(* PLC project mtcs_m2, Institute of Astronomy OntoManager 0.0.1 *)
(* stored: creationDateTime 2017-02-03T09:55:41.735679, modificationDateTime 2017-02-03T09:55:41.735679 *)

TYPE M2Axes : (X := 0, Y := 1, Z := 2, TILTX := 3, TILTY := 4);
END_TYPE

TYPE M2MoveProcedureStates : (IDLE := 0, ABORTED := 1, PREPARE_PROCESS := 2, MOVING := 3, MOVING_TO_ANTI_BACKLASH_POSITION := 4, MOVING_CLOSE_TO_FINAL_POSITION := 5, MOVING_TO_FINAL_POSITION := 6, ERROR := 7, ABORTING := 8);
END_TYPE

TYPE M2Parts : STRUCT
  powerRelay : SimpleRelay;  (* Relay to power on/off the power of the M2 field electricity *)
  heater : SimpleRelay;  (* Digital output to power on/off the heater of M2 *)
  x : M2XAxis;  (* The X axis *)
  y : M2YAxis;  (* The Y axis *)
  z : M2ZAxis;  (* The Z axis *)
  tiltX : M2TiltXAxis;  (* The TiltX axis *)
  tiltY : M2TiltYAxis;  (* The TiltY axis *)
  multiplexer : M2Multiplexer;  (* The multiplexer inputs and outputs *)
  configManager : ConfigManager;  (* The config manager (to load/save/activate configuration data) *)
  moveStepsProcedure : M2MoveStepsProcedure;  (* The move steps procedure *)
  movePositionProcedure : M2MovePositionProcedure;  (* The move to a certain position procedure *)
END_STRUCT;
END_TYPE

TYPE M2MultiplexerParts : STRUCT
  A : SimpleRelay;  (* Output A of the multiplexer corresponding with the selected axis *)
  B : SimpleRelay;  (* Output B of the multiplexer corresponding with the selected axis *)
  C : SimpleRelay;  (* Output C of the multiplexer corresponding with the selected axis *)
  driveEnable : SimpleRelay;  (* Enabled (TRUE) if the drive selected by the multiplexer must be enabled, Disabled (FALSE) if it must be disabled *)
  CW : SimpleRelay;  (* Enabled (TRUE) if the motor selected by the multiplexer will run in CW direction (- motion on the screw), Disabled (FALSE) if it will run in CCW direction (+ motion on the screw) *)
  release : SimpleRelay;  (* Disabled (FALSE) if the motor selected by the multiplexer must be braking, Enabled (TRUE) if it must be released *)
END_STRUCT;
END_TYPE

TYPE M2ZAxisParts : STRUCT
  highSpeed : SimpleRelay;  (* Enabled (TRUE) to enable the high-speed motion of the Z axis, Disabled (FALSE) to leave it low-speed *)
  encoder : SSIEncoder;  (* The SSI encoder of the Z axis *)
END_STRUCT;
END_TYPE

TYPE M2Processes : STRUCT
  initialize : Process;  (* Start initializing *)
  lock : Process;  (* Lock the system *)
  unlock : Process;  (* Unlock the system *)
  changeOperatingState : ChangeOperatingStateProcess;  (* Change the operating state (e.g. AUTO, MANUAL, ...) *)
  moveAbsolute : M2MoveProcess;  (* Move the position of one axis in an absolute way *)
  moveRelative : M2MoveProcess;  (* Move the position of one axis relative to the current position *)
  moveSteps : M2MoveStepsProcess;  (* Move the position of one axis by providing a number of steps (i.e. motor pulses) *)
  doThermalFocus : Process;  (* Do a thermal focus for the currently active focus *)
  doThermalFocusForStationName : M2DoThermalFocusForStationName;  (* Do a thermal focus for a specified focal station (based on the configured name of the station) *)
  doThermalFocusForStationPosition : M2DoThermalFocusForStationPosition;  (* Do a thermal focus for a specified focal station (based on the station numerical ID) *)
  verifyFixedPositions : Process;  (* Verify (and adjust if necessary) the fixed positions of X, Y, TiltX, and TiltY *)
  powerOn : Process;  (* Power on the M2 electricity *)
  powerOff : Process;  (* Power off the M2 electricity *)
  abort : Process;  (* Abort the move procedure *)
END_STRUCT;
END_TYPE

TYPE M2MultiplexerProcesses : STRUCT
  selectAxis : M2SelectAxisProcess;  (* Select an axis *)
END_STRUCT;
END_TYPE

TYPE M2Statuses : STRUCT
  initializationStatus : InitializationStatus;
  poweredStatus : PoweredStatus;
  healthStatus : HealthStatus;
  busyStatus : BusyStatus;
  operatingStatus : OperatingStatus;
END_STRUCT;
END_TYPE

TYPE M2MultiplexerStatuses : STRUCT
  healthStatus : HealthStatus;  (* Is the selected drive healthy? *)
  busyStatus : BusyStatus;  (* Is the selected drive busy? *)
END_STRUCT;
END_TYPE

TYPE M2XAxisStatuses : STRUCT
  healthStatus : HealthStatus;  (* Is the axis healthy? *)
END_STRUCT;
END_TYPE

TYPE M2YAxisStatuses : STRUCT
  healthStatus : HealthStatus;  (* Is the axis healthy? *)
END_STRUCT;
END_TYPE

TYPE M2TiltXAxisStatuses : STRUCT
  healthStatus : HealthStatus;  (* Is the axis healthy? *)
END_STRUCT;
END_TYPE

TYPE M2TiltYAxisStatuses : STRUCT
  healthStatus : HealthStatus;  (* Is the axis healthy? *)
END_STRUCT;
END_TYPE

TYPE M2ZAxisStatuses : STRUCT
  healthStatus : HealthStatus;  (* Is the axis healthy? *)
END_STRUCT;
END_TYPE

TYPE M2MoveStepsProcedureStatuses : STRUCT
  busyStatus : BusyStatus;  (* Is the M2MoveStepsProcedure in a busy state? *)
  healthStatus : HealthStatus;  (* Is the M2MoveStepsProcedure in a healthy state? *)
END_STRUCT;
END_TYPE

TYPE M2MovePositionProcedureStatuses : STRUCT
  busyStatus : BusyStatus;  (* Is the M2MoveAbsoluteProcedure in a busy state? *)
  healthStatus : HealthStatus;  (* Is the M2MoveAbsoluteProcedure in a healthy state? *)
END_STRUCT;
END_TYPE

TYPE M2Config : STRUCT
  x : M2PotentiometerAxisConfig;  (* The config of the X axis *)
  y : M2PotentiometerAxisConfig;  (* The config of the Y axis *)
  z : M2ZAxisConfig;  (* The config of the Z axis *)
  tiltX : M2PotentiometerAxisConfig;  (* The config of the tiltX axis *)
  tiltY : M2PotentiometerAxisConfig;  (* The config of the tiltY axis *)
  thermalFocus : M2ThermalFocusConfig;  (* The thermal focus coefficients for all focal stations *)
  waitAfterPowerOn : LREAL;  (* Time (in seconds) to wait after the field electricity of M2 have been powered on *)
  waitAfterPowerOff : LREAL;  (* Time (in seconds) to wait after the field electricity of M2 have been powered off *)
  powerOffTimeout : LREAL;  (* If no new command is sent to M2 within this time (in seconds) after completion of the last command, M2 will be powered off automatically *)
  fixedXPosition : LREAL;  (* The fixed X position in mm *)
  fixedXPositionTolerance : LREAL;  (* If the X position is within fixedXPosition +/- this tolerance, there's no need to adjust it *)
  fixedYPosition : LREAL;  (* The fixed Y position in mm *)
  fixedYPositionTolerance : LREAL;  (* If the Y position is within fixedYPosition +/- this tolerance, there's no need to adjust it *)
  fixedTiltXPosition : LREAL;  (* The fixed TiltX position in mm *)
  fixedTiltXPositionTolerance : LREAL;  (* If the TiltX position is within fixedTiltXPosition +/- this tolerance, there's no need to adjust it *)
  fixedTiltYPosition : LREAL;  (* The fixed TiltY position in mm *)
  fixedTiltYPositionTolerance : LREAL;  (* If the TiltY position is within fixedTiltYPosition +/- this tolerance, there's no need to adjust it *)
  verifyFixedPositinsOnThermalFocus : BOOL;  (* Each time a theremal focus is done, verify the fixed positions (and adjust them if they fall out of the tolerance) *)
END_STRUCT;
END_TYPE

TYPE M2ThermalFocusStationConfig : STRUCT
  offset : LREAL;  (* focus = offset + topCoefficient*topTemperature + centreCoefficient*centreTemperature + mirrorCellCoefficient*mirrorCellTemperature *)
  topCoefficient : LREAL;  (* focus = offset + topCoefficient*topTemperature + centreCoefficient*centreTemperature + mirrorCellCoefficient*mirrorCellTemperature *)
  centreCoefficient : LREAL;  (* focus = offset + topCoefficient*topTemperature + centreCoefficient*centreTemperature + mirrorCellCoefficient*mirrorCellTemperature *)
  mirrorCellCoefficient : LREAL;  (* focus = offset + topCoefficient*topTemperature + centreCoefficient*centreTemperature + mirrorCellCoefficient*mirrorCellTemperature *)
END_STRUCT;
END_TYPE

TYPE M2ThermalFocusConfig : STRUCT
  cassegrain : M2ThermalFocusStationConfig;  (* Cassegrain thermal focus config *)
  nasmythA : M2ThermalFocusStationConfig;  (* Nasmyth A thermal focus config *)
  nasmythB : M2ThermalFocusStationConfig;  (* Nasmyth B thermal focus config *)
  nasmythC : M2ThermalFocusStationConfig;  (* Nasmyth C thermal focus config *)
  nasmythD : M2ThermalFocusStationConfig;  (* Nasmyth D thermal focus config *)
  other0 : M2ThermalFocusStationConfig;  (* Other 0 thermal focus config *)
  other1 : M2ThermalFocusStationConfig;  (* Other 1 thermal focus config *)
  other2 : M2ThermalFocusStationConfig;  (* Other 2 thermal focus config *)
  other3 : M2ThermalFocusStationConfig;  (* Other 3 thermal focus config *)
  other4 : M2ThermalFocusStationConfig;  (* Other 4 thermal focus config *)
END_STRUCT;
END_TYPE

TYPE M2AxisGeneralConfig : STRUCT
  measurement : MeasurementConfig;  (* Configure the position measurement *)
  stoppingSteps : UDINT;  (* The number of steps to be expected between the time at which the PLC realizes that the brake release signal must be set, and the time that the axis is fully stopped (for Z axis: at low speed) *)
  finalSenseCW : BOOL;  (* TRUE if the motor final sense must be ClockWise (- motion on the screw), FALSE if the motor final sense must be CounterClockWise (+ motion on the screw) (for Z axis: at low speed) *)
  closePosition : UDINT;  (* The number of steps between the Close position (C) and final position (F) *)
  antiBacklashPosition : UDINT;  (* The number of steps between the Anti-backlash position (A) and final position (F) *)
  waitAfterMove : LREAL;  (* Time (in seconds) to wait after the axis has been moved *)
  timeout : LREAL;  (* Timeout for a movement, in seconds (for Z-axis: at low speed) *)
END_STRUCT;
END_TYPE

TYPE M2ZAxisConfig : STRUCT
  general : M2AxisGeneralConfig;  (* Settings which are general for all axes *)
  highSpeedStoppingSteps : UDINT;  (* The number of steps to be expected between the time at which the PLC realizes that the brake release signal must be set, and the time that the axis is fully stopped at high speed *)
  highSpeedTimeout : LREAL;  (* Timeout for a fast movement of the Z axis (in seconds) *)
END_STRUCT;
END_TYPE

TYPE M2PotentiometerAxisConfig : STRUCT
  general : M2AxisGeneralConfig;  (* Settings which are general for all axes *)
  voltageCorrectionFactor : LREAL;  (* Position = voltage * correctionFactor * voltageToPosition *)
END_STRUCT;
END_TYPE

TYPE M2ConstantsZ : STRUCT
  MOT_TO_RED_RATIO : LREAL := 134.0;  (* Motor reduction ratio *)
  RED_TO_SCREW_RATIO : LREAL := 2.0;  (* Transmission ratio between the motor reduction and the screw *)
  SCREW_TO_ENC_RATIO : LREAL := 1.0;  (* Transmission ratio between the encoder and the screw *)
  MIN_POSITION : LREAL := 0.0;  (* Minimum position of the axis, in micrometer *)
  MAX_POSITION : LREAL := 50000.0;  (* Maximum position of the axis, in micrometer *)
  SCREW_PITCH : LREAL := 2000.0;  (* Screw pitch, in micrometer *)
  FEEDBACK_RESOLUTION : LREAL := 32;  (* Motor feedback resolution (pulses per revolution of the motor rotor) *)
END_STRUCT;
END_TYPE

TYPE M2ConstantsX : STRUCT
  MOT_TO_RED_RATIO : LREAL := 415.0;  (* Motor reduction ratio *)
  RED_TO_SCREW_RATIO : LREAL := 2.0;  (* Transmission ratio between the motor reduction and the screw *)
  SCREW_TO_POT_RATIO : LREAL := 0.5;  (* Transmission ratio between the potentiometer and the screw *)
  MIN_POSITION : LREAL := 400.0;  (* Minimum position of the axis, in micrometer *)
  MAX_POSITION : LREAL := 4700.0;  (* Maximum position of the axis, in micrometer *)
  SCREW_PITCH : LREAL := 1000.0;  (* Screw pitch, in micrometer *)
  FEEDBACK_RESOLUTION : LREAL := 3;  (* Motor feedback resolution (pulses per revolution of the motor rotor) *)
  POTENTIOMETER_REVOLUTIONS : LREAL := 10;  (* Max number of revolutions of the potentiometer *)
END_STRUCT;
END_TYPE

TYPE M2ConstantsY : STRUCT
  MOT_TO_RED_RATIO : LREAL := 415.0;  (* Motor reduction ratio *)
  RED_TO_SCREW_RATIO : LREAL := 2.0;  (* Transmission ratio between the motor reduction and the screw *)
  SCREW_TO_POT_RATIO : LREAL := 0.5;  (* Transmission ratio between the potentiometer and the screw *)
  MIN_POSITION : LREAL := 400.0;  (* Minimum position of the axis, in micrometer *)
  MAX_POSITION : LREAL := 4700.0;  (* Maximum position of the axis, in micrometer *)
  SCREW_PITCH : LREAL := 1000.0;  (* Screw pitch, in micrometer *)
  FEEDBACK_RESOLUTION : LREAL := 3;  (* Motor feedback resolution (pulses per revolution of the motor rotor) *)
  POTENTIOMETER_REVOLUTIONS : LREAL := 10;  (* Max number of revolutions of the potentiometer *)
END_STRUCT;
END_TYPE

TYPE M2ConstantsTiltX : STRUCT
  MOT_TO_RED_RATIO : LREAL := 1526.0;  (* Motor reduction ratio *)
  RED_TO_SCREW_RATIO : LREAL := 2.0;  (* Transmission ratio between the motor reduction and the screw *)
  SCREW_TO_POT_RATIO : LREAL := 0.5;  (* Transmission ratio between the potentiometer and the screw *)
  MIN_POSITION : LREAL := 260.0;  (* Minimum position of the axis, in micrometer *)
  MAX_POSITION : LREAL := 1200.0;  (* Maximum position of the axis, in micrometer *)
  SCREW_PITCH : LREAL := 1000.0;  (* Screw pitch, in micrometer *)
  FEEDBACK_RESOLUTION : LREAL := 3;  (* Motor feedback resolution (pulses per revolution of the motor rotor) *)
  POTENTIOMETER_REVOLUTIONS : LREAL := 3;  (* Max number of revolutions of the potentiometer *)
END_STRUCT;
END_TYPE

TYPE M2ConstantsTiltY : STRUCT
  MOT_TO_RED_RATIO : LREAL := 1526.0;  (* Motor reduction ratio *)
  RED_TO_SCREW_RATIO : LREAL := 2.0;  (* Transmission ratio between the motor reduction and the screw *)
  SCREW_TO_POT_RATIO : LREAL := 0.5;  (* Transmission ratio between the potentiometer and the screw *)
  MIN_POSITION : LREAL := 180.0;  (* Minimum position of the axis, in micrometer *)
  MAX_POSITION : LREAL := 1200.0;  (* Maximum position of the axis, in micrometer *)
  SCREW_PITCH : LREAL := 1000.0;  (* Screw pitch, in micrometer *)
  FEEDBACK_RESOLUTION : LREAL := 3;  (* Motor feedback resolution (pulses per revolution of the motor rotor) *)
  POTENTIOMETER_REVOLUTIONS : LREAL := 3;  (* Max number of revolutions of the potentiometer *)
END_STRUCT;
END_TYPE

TYPE M2SelectAxisProcessArgs : STRUCT
  axis : M2Axes;  (* The axis to select *)
END_STRUCT;
END_TYPE

TYPE M2MoveProcessArgs : STRUCT
  axis : M2Axes;  (* The axis to move *)
  position : LREAL;  (* Move to a certain position in millimeters *)
END_STRUCT;
END_TYPE

TYPE M2MoveStepsProcessArgs : STRUCT
  axis : M2Axes;  (* The axis to move *)
  steps : UDINT;  (* Move a certain number of steps *)
  cw : BOOL;  (* True if the axis should be moved in CW (negative) direction *)
  fast : BOOL;  (* True if the axis should be moved fast (only used in case of Z-axis!) *)
END_STRUCT;
END_TYPE

TYPE M2DoThermalFocusForStationPositionArgs : STRUCT
  station : M3PositionIDs;  (* The station numerical ID for which the thermal focus should be executed *)
END_STRUCT;
END_TYPE

TYPE M2DoThermalFocusForStationNameArgs : STRUCT
  station : STRING;  (* The configured station name, for which the thermal focus should be executed *)
END_STRUCT;
END_TYPE

FUNCTION_BLOCK SM_M2
  VAR_INPUT
    {attribute 'OPC.UA.DA' := '1'}
    {attribute 'OPC.UA.DA.Access' := '1'}
    editableConfig : M2Config;  (* Editable configuration of the M2 subsystem *)
  END_VAR
  VAR_OUTPUT
    {attribute 'OPC.UA.DA' := '1'}
    {attribute 'OPC.UA.DA.Access' := '1'}
    actualStatus : STRING;  (* Current status description *)
    previousStatus : STRING;  (* Previous status description *)
    {attribute 'OPC.UA.DA' := '1'}
    {attribute 'OPC.UA.DA.Access' := '1'}
    config : M2Config;  (* Active configuration of the M2 subsystem *)
    {attribute 'OPC.UA.DA' := '1'}
    {attribute 'OPC.UA.DA.Access' := '1'}
    selectedAxis : M2Axes;  (* The axis which is currently selected by the multiplexer *)
    {attribute 'OPC.UA.DA' := '1'}
    {attribute 'OPC.UA.DA.Access' := '1'}
    selectedAxisName : STRING;  (* The name of the axis which is currently selected by the multiplexer *)
    {attribute 'OPC.UA.DA' := '1'}
    {attribute 'OPC.UA.DA.Access' := '1'}
    powerOffTimer : LREAL;  (* Number of seconds before the power of the M2 field electricity will be powered off automatically *)
    {attribute 'OPC.UA.DA' := '1'}
    {attribute 'OPC.UA.DA.Access' := '1'}
    thermalFocusCassegrain : LinearPosition;  (* Thermal focus position for cassegrain *)
    {attribute 'OPC.UA.DA' := '1'}
    {attribute 'OPC.UA.DA.Access' := '1'}
    thermalFocusNasmythA : LinearPosition;  (* Thermal focus position for nasmyth A *)
    {attribute 'OPC.UA.DA' := '1'}
    {attribute 'OPC.UA.DA.Access' := '1'}
    thermalFocusNasmythB : LinearPosition;  (* Thermal focus position for nasmyth B *)
    {attribute 'OPC.UA.DA' := '1'}
    {attribute 'OPC.UA.DA.Access' := '1'}
    thermalFocusNasmythC : LinearPosition;  (* Thermal focus position for nasmyth C *)
    {attribute 'OPC.UA.DA' := '1'}
    {attribute 'OPC.UA.DA.Access' := '1'}
    thermalFocusNasmythD : LinearPosition;  (* Thermal focus position for nasmyth D *)
    {attribute 'OPC.UA.DA' := '1'}
    {attribute 'OPC.UA.DA.Access' := '1'}
    thermalFocusActualFocalStation : LinearPosition;  (* Thermal focus position for nasmyth D *)
    statuses : M2Statuses;  (* Statuses of the state machine *)
    parts : M2Parts;  (* Parts of the state machine *)
    processes : M2Processes;  (* Processes of the state machine *)
  END_VAR
  VAR_IN_OUT
    {attribute 'OPC.UA.DA' := '0'}
    operatorStatus : OperatorStatus;  (* Shared operator status *)
    {attribute 'OPC.UA.DA' := '0'}
    io : M1M2IO;  (* Shared I/O with M1 *)
    {attribute 'OPC.UA.DA' := '0'}
    actualFocalStation : M3PositionIDs;  (* Actual M3 focal station, needed for thermal focus *)
    {attribute 'OPC.UA.DA' := '0'}
    m3KnownPositionsConfig : M3KnownPositionsConfig;  (* Config of M3 with all info (e.g. names) of focal stations *)
    {attribute 'OPC.UA.DA' := '0'}
    temperatures : TelemetryTemperatures;  (* Telemetry temperatures *)
  END_VAR

            parts.powerRelay( isEnabled := operatorStatus.tech );
parts.heater( isEnabled := operatorStatus.tech );
parts.x(
    powered := statuses.poweredStatus.enabled,
    config := config,
    axisConfig := config.x);
parts.y(
    powered := statuses.poweredStatus.enabled,
    config := config,
    axisConfig := config.y);
parts.z(
    powered := statuses.poweredStatus.enabled,
    config := config,
    axisConfig := config.z,
    isEnabled := operatorStatus.tech);
parts.tiltX(
    powered := statuses.poweredStatus.enabled,
    config := config,
    axisConfig := config.tiltX);
parts.tiltY(
    powered := statuses.poweredStatus.enabled,
    config := config,
    axisConfig := config.tiltY);
parts.multiplexer(
    isEnabled := operatorStatus.tech,
    powered := statuses.poweredStatus.enabled);
parts.configManager( isEnabled := operatorStatus.tech );
parts.moveStepsProcedure(
    powerOn := processes.powerOn,
    x := parts.x,
    y := parts.y,
    z := parts.z,
    tiltX := parts.tiltX,
    tiltY := parts.tiltY,
    multiplexer := parts.multiplexer,
    config := config);
parts.movePositionProcedure(
    powerOn := processes.powerOn,
    x := parts.x,
    y := parts.y,
    z := parts.z,
    tiltX := parts.tiltX,
    tiltY := parts.tiltY,
    multiplexer := parts.multiplexer,
    moveStepsProcedure := parts.moveStepsProcedure,
    config := config);
statuses.initializationStatus();
statuses.poweredStatus( isEnabled := parts.powerRelay.digitalOutput AND (processes.powerOn.statuses.busyStatus.idle AND processes.powerOff.statuses.busyStatus.idle) );
statuses.healthStatus(
    isGood := ((parts.x.statuses.healthStatus.isGood AND (parts.y.statuses.healthStatus.isGood AND (parts.z.statuses.healthStatus.isGood AND (parts.tiltX.statuses.healthStatus.isGood AND (parts.tiltY.statuses.healthStatus.isGood AND parts.multiplexer.statuses.healthStatus.isGood))))) OR statuses.poweredStatus.disabled) AND (io.statuses.healthStatus.isGood AND (temperatures.statuses.healthStatus.isGood AND parts.configManager.statuses.healthStatus.isGood)),
    hasWarning := ((parts.x.statuses.healthStatus.hasWarning OR (parts.y.statuses.healthStatus.hasWarning OR (parts.z.statuses.healthStatus.hasWarning OR (parts.tiltX.statuses.healthStatus.hasWarning OR (parts.tiltY.statuses.healthStatus.hasWarning OR parts.multiplexer.statuses.healthStatus.hasWarning))))) AND statuses.poweredStatus.enabled) OR (io.statuses.healthStatus.hasWarning OR (temperatures.statuses.healthStatus.hasWarning OR parts.configManager.statuses.healthStatus.hasWarning)));
statuses.busyStatus( isBusy := statuses.initializationStatus.initializing OR (parts.multiplexer.statuses.busyStatus.busy OR (parts.configManager.statuses.busyStatus.busy OR (processes.abort.statuses.busyStatus.busy OR (processes.powerOn.statuses.busyStatus.busy OR (processes.powerOff.statuses.busyStatus.busy OR (processes.doThermalFocus.statuses.busyStatus.busy OR (processes.doThermalFocusForStationName.statuses.busyStatus.busy OR (processes.doThermalFocusForStationPosition.statuses.busyStatus.busy OR (processes.verifyFixedPositions.statuses.busyStatus.busy OR (processes.moveSteps.statuses.busyStatus.busy OR (processes.moveAbsolute.statuses.busyStatus.busy OR processes.moveRelative.statuses.busyStatus.busy))))))))))) );
statuses.operatingStatus( superState := statuses.initializationStatus.initialized );
processes.initialize( isEnabled := statuses.initializationStatus.shutdown OR (statuses.initializationStatus.initializingFailed OR statuses.initializationStatus.initialized) );
processes.lock( isEnabled := operatorStatus.tech AND statuses.initializationStatus.initialized );
processes.unlock( isEnabled := operatorStatus.tech AND statuses.initializationStatus.locked );
processes.changeOperatingState( isEnabled := statuses.busyStatus.idle AND (statuses.initializationStatus.initialized AND operatorStatus.tech) );
processes.moveAbsolute( isEnabled := statuses.initializationStatus.initialized AND statuses.busyStatus.idle );
processes.moveRelative( isEnabled := processes.moveAbsolute.isEnabled );
processes.moveSteps( isEnabled := statuses.initializationStatus.initialized AND operatorStatus.tech );
processes.doThermalFocus( isEnabled := processes.moveAbsolute.isEnabled AND (NOT(actualFocalStation = M3PositionIDs.UNKNOWN)) );
processes.doThermalFocusForStationName( isEnabled := processes.moveAbsolute.isEnabled );
processes.doThermalFocusForStationPosition( isEnabled := processes.moveAbsolute.isEnabled );
processes.verifyFixedPositions( isEnabled := processes.moveAbsolute.isEnabled );
processes.powerOn( isEnabled := statuses.busyStatus.idle AND statuses.initializationStatus.initialized );
processes.powerOff( isEnabled := statuses.busyStatus.idle AND statuses.initializationStatus.initialized );
processes.abort( isEnabled := parts.moveStepsProcedure.statuses.busyStatus.busy OR parts.movePositionProcedure.statuses.busyStatus.busy );

          

{attribute 'TcRpcEnable' := '1'}
METHOD initialize : RequestResults
                  initialize := THIS^.processes.initialize.request();

                
END_METHOD

{attribute 'TcRpcEnable' := '1'}
METHOD lock : RequestResults
                  lock := THIS^.processes.lock.request();

                
END_METHOD

{attribute 'TcRpcEnable' := '1'}
METHOD unlock : RequestResults
                  unlock := THIS^.processes.unlock.request();

                
END_METHOD

{attribute 'TcRpcEnable' := '1'}
METHOD changeOperatingState : RequestResults
  VAR_INPUT
    state : OperatingStates;
  END_VAR
                  changeOperatingState := THIS^.processes.changeOperatingState.request( state := state );

                
END_METHOD

{attribute 'TcRpcEnable' := '1'}
METHOD moveAbsolute : RequestResults
  VAR_INPUT
    axis : M2Axes;
    position : LREAL;
  END_VAR
                  moveAbsolute := THIS^.processes.moveAbsolute.request(
    axis := axis,
    position := position);

                
END_METHOD

{attribute 'TcRpcEnable' := '1'}
METHOD moveRelative : RequestResults
  VAR_INPUT
    axis : M2Axes;
    position : LREAL;
  END_VAR
                  moveRelative := THIS^.processes.moveRelative.request(
    axis := axis,
    position := position);

                
END_METHOD

{attribute 'TcRpcEnable' := '1'}
METHOD moveSteps : RequestResults
  VAR_INPUT
    axis : M2Axes;
    steps : UDINT;
    cw : BOOL;
    fast : BOOL;
  END_VAR
                  moveSteps := THIS^.processes.moveSteps.request(
    axis := axis,
    steps := steps,
    cw := cw,
    fast := fast);

                
END_METHOD

{attribute 'TcRpcEnable' := '1'}
METHOD doThermalFocus : RequestResults
                  doThermalFocus := THIS^.processes.doThermalFocus.request();

                
END_METHOD

{attribute 'TcRpcEnable' := '1'}
METHOD doThermalFocusForStationName : RequestResults
  VAR_INPUT
    station : STRING;
  END_VAR
                  doThermalFocusForStationName := THIS^.processes.doThermalFocusForStationName.request( station := station );

                
END_METHOD

{attribute 'TcRpcEnable' := '1'}
METHOD doThermalFocusForStationPosition : RequestResults
  VAR_INPUT
    station : M3PositionIDs;
  END_VAR
                  doThermalFocusForStationPosition := THIS^.processes.doThermalFocusForStationPosition.request( station := station );

                
END_METHOD

{attribute 'TcRpcEnable' := '1'}
METHOD verifyFixedPositions : RequestResults
                  verifyFixedPositions := THIS^.processes.verifyFixedPositions.request();

                
END_METHOD

{attribute 'TcRpcEnable' := '1'}
METHOD powerOn : RequestResults
                  powerOn := THIS^.processes.powerOn.request();

                
END_METHOD

{attribute 'TcRpcEnable' := '1'}
METHOD powerOff : RequestResults
                  powerOff := THIS^.processes.powerOff.request();

                
END_METHOD

{attribute 'TcRpcEnable' := '1'}
METHOD abort : RequestResults
                  abort := THIS^.processes.abort.request();

                
END_METHOD

{attribute 'TcRpcEnable' := '1'}
METHOD _log : BOOL
  VAR_INPUT
    name : STRING;  (* Name of this function block instance *)
  END_VAR
  VAR_IN_OUT
    buffer : LogBuffer;  (* Buffer to write all logging to *)
  END_VAR
  VAR
    subBuffer : LogBuffer;  (* Temporary buffer to write logging by parts (sub-statemachines) to *)
  END_VAR
                  THIS^.parts.powerRelay._log(
    name := 'powerRelay',
    buffer := subBuffer);
THIS^.parts.heater._log(
    name := 'heater',
    buffer := subBuffer);
THIS^.parts.x._log(
    name := 'x',
    buffer := subBuffer);
THIS^.parts.y._log(
    name := 'y',
    buffer := subBuffer);
THIS^.parts.z._log(
    name := 'z',
    buffer := subBuffer);
THIS^.parts.tiltX._log(
    name := 'tiltX',
    buffer := subBuffer);
THIS^.parts.tiltY._log(
    name := 'tiltY',
    buffer := subBuffer);
THIS^.parts.multiplexer._log(
    name := 'multiplexer',
    buffer := subBuffer);
THIS^.parts.configManager._log(
    name := 'configManager',
    buffer := subBuffer);
THIS^.parts.moveStepsProcedure._log(
    name := 'moveStepsProcedure',
    buffer := subBuffer);
THIS^.parts.movePositionProcedure._log(
    name := 'movePositionProcedure',
    buffer := subBuffer);
LOGGER(
    name := name,
    actualStatus := THIS^.actualStatus,
    previousStatus := THIS^.previousStatus,
    buffer := buffer,
    subBuffer := subBuffer,
    pHealthStatus := ADR(THIS^.statuses.healthStatus),
    pBusyStatus := ADR(THIS^.statuses.busyStatus));

                
END_METHOD
END_FUNCTION_BLOCK

FUNCTION_BLOCK SM_M2Multiplexer
  VAR_INPUT
    {attribute 'OPC.UA.DA' := '1'}
    {attribute 'OPC.UA.DA.Access' := '1'}
    noFault AT %I* : BOOL;  (* FALSE if the drive selected by the multiplexer is in faulty state, TRUE if it is in a healthy state *)
    {attribute 'OPC.UA.DA' := '1'}
    {attribute 'OPC.UA.DA.Access' := '1'}
    isEnabled : BOOL;  (* TRUE if the multiplexer is enabled, FALSE if not *)
    {attribute 'OPC.UA.DA' := '1'}
    {attribute 'OPC.UA.DA.Access' := '1'}
    powered : BOOL;  (* TRUE if the axis is powered *)
  END_VAR
  VAR_OUTPUT
    {attribute 'OPC.UA.DA' := '1'}
    {attribute 'OPC.UA.DA.Access' := '1'}
    actualStatus : STRING;  (* Current status description *)
    previousStatus : STRING;  (* Previous status description *)
    statuses : M2MultiplexerStatuses;  (* Statuses of the state machine *)
    parts : M2MultiplexerParts;  (* Parts of the state machine *)
    processes : M2MultiplexerProcesses;  (* Processes of the state machine *)
  END_VAR

            parts.A( isEnabled := isEnabled );
parts.B( isEnabled := isEnabled );
parts.C( isEnabled := isEnabled );
parts.driveEnable( isEnabled := isEnabled );
parts.CW( isEnabled := isEnabled );
parts.release( isEnabled := isEnabled );
statuses.healthStatus( isGood := (noFault OR (NOT(powered))) AND processes.selectAxis.statuses.healthStatus.good );
statuses.busyStatus( isBusy := parts.A.statuses.busyStatus.busy OR (parts.B.statuses.busyStatus.busy OR (parts.C.statuses.busyStatus.busy OR (parts.driveEnable.statuses.busyStatus.busy OR (parts.CW.statuses.busyStatus.busy OR parts.release.statuses.busyStatus.busy)))) );
processes.selectAxis( isEnabled := isEnabled );

          

{attribute 'TcRpcEnable' := '1'}
METHOD selectAxis : RequestResults
  VAR_INPUT
    axis : M2Axes;
  END_VAR
                  selectAxis := THIS^.processes.selectAxis.request( axis := axis );

                
END_METHOD

{attribute 'TcRpcEnable' := '1'}
METHOD _log : BOOL
  VAR_INPUT
    name : STRING;  (* Name of this function block instance *)
  END_VAR
  VAR_IN_OUT
    buffer : LogBuffer;  (* Buffer to write all logging to *)
  END_VAR
  VAR
    subBuffer : LogBuffer;  (* Temporary buffer to write logging by parts (sub-statemachines) to *)
  END_VAR
                  THIS^.parts.A._log(
    name := 'A',
    buffer := subBuffer);
THIS^.parts.B._log(
    name := 'B',
    buffer := subBuffer);
THIS^.parts.C._log(
    name := 'C',
    buffer := subBuffer);
THIS^.parts.driveEnable._log(
    name := 'driveEnable',
    buffer := subBuffer);
THIS^.parts.CW._log(
    name := 'CW',
    buffer := subBuffer);
THIS^.parts.release._log(
    name := 'release',
    buffer := subBuffer);
LOGGER(
    name := name,
    actualStatus := THIS^.actualStatus,
    previousStatus := THIS^.previousStatus,
    buffer := buffer,
    subBuffer := subBuffer,
    pHealthStatus := ADR(THIS^.statuses.healthStatus),
    pBusyStatus := ADR(THIS^.statuses.busyStatus));

                
END_METHOD
END_FUNCTION_BLOCK

FUNCTION_BLOCK SM_M2XAxis
  VAR_INPUT
    {attribute 'OPC.UA.DA' := '1'}
    {attribute 'OPC.UA.DA.Access' := '1'}
    position : LinearPositionMeasurement16;  (* Actual position of the axis *)
    {attribute 'OPC.UA.DA' := '1'}
    {attribute 'OPC.UA.DA.Access' := '1'}
    backlashLifted : BOOL;  (* TRUE if the backlash was previously lifted *)
    {attribute 'OPC.UA.DA' := '1'}
    {attribute 'OPC.UA.DA.Access' := '1'}
    powered : BOOL;  (* TRUE if the axis is powered *)
  END_VAR
  VAR_OUTPUT
    {attribute 'OPC.UA.DA' := '1'}
    {attribute 'OPC.UA.DA.Access' := '1'}
    actualStatus : STRING;  (* Current status description *)
    previousStatus : STRING;  (* Previous status description *)
    {attribute 'OPC.UA.DA' := '1'}
    {attribute 'OPC.UA.DA.Access' := '1'}
    constants : M2ConstantsX;  (* Some constants particular for this axis *)
    statuses : M2XAxisStatuses;  (* Statuses of the state machine *)
  END_VAR
  VAR_IN_OUT
    {attribute 'OPC.UA.DA' := '0'}
    config : M2Config;  (* The general M2 config *)
    {attribute 'OPC.UA.DA' := '0'}
    axisConfig : M2PotentiometerAxisConfig;  (* The config particular for this axis *)
  END_VAR

            position(
    config := axisConfig.general.measurement,
    conversionFactor := (constants.POTENTIOMETER_REVOLUTIONS * (constants.SCREW_TO_POT_RATIO * constants.SCREW_PITCH)) / (32768.0 * 1000.0));
statuses.healthStatus(
    isGood := position.statuses.healthStatus.isGood,
    hasWarning := position.statuses.healthStatus.hasWarning);

          

{attribute 'TcRpcEnable' := '1'}
METHOD _log : BOOL
  VAR_INPUT
    name : STRING;  (* Name of this function block instance *)
  END_VAR
  VAR_IN_OUT
    buffer : LogBuffer;  (* Buffer to write all logging to *)
  END_VAR
  VAR
    subBuffer : LogBuffer;  (* Temporary buffer to write logging by parts (sub-statemachines) to *)
  END_VAR
                  LOGGER(
    name := name,
    actualStatus := THIS^.actualStatus,
    previousStatus := THIS^.previousStatus,
    buffer := buffer,
    subBuffer := subBuffer,
    pHealthStatus := ADR(THIS^.statuses.healthStatus));

                
END_METHOD
END_FUNCTION_BLOCK

FUNCTION_BLOCK SM_M2YAxis
  VAR_INPUT
    {attribute 'OPC.UA.DA' := '1'}
    {attribute 'OPC.UA.DA.Access' := '1'}
    position : LinearPositionMeasurement16;  (* Actual position of the axis *)
    {attribute 'OPC.UA.DA' := '1'}
    {attribute 'OPC.UA.DA.Access' := '1'}
    backlashLifted : BOOL;  (* TRUE if the backlash was previously lifted *)
    {attribute 'OPC.UA.DA' := '1'}
    {attribute 'OPC.UA.DA.Access' := '1'}
    powered : BOOL;  (* TRUE if the axis is powered *)
  END_VAR
  VAR_OUTPUT
    {attribute 'OPC.UA.DA' := '1'}
    {attribute 'OPC.UA.DA.Access' := '1'}
    actualStatus : STRING;  (* Current status description *)
    previousStatus : STRING;  (* Previous status description *)
    {attribute 'OPC.UA.DA' := '1'}
    {attribute 'OPC.UA.DA.Access' := '1'}
    constants : M2ConstantsY;  (* Some constants particular for this axis *)
    statuses : M2YAxisStatuses;  (* Statuses of the state machine *)
  END_VAR
  VAR_IN_OUT
    {attribute 'OPC.UA.DA' := '0'}
    config : M2Config;  (* The general M2 config *)
    {attribute 'OPC.UA.DA' := '0'}
    axisConfig : M2PotentiometerAxisConfig;  (* The config particular for this axis *)
  END_VAR

            position(
    config := axisConfig.general.measurement,
    conversionFactor := (constants.POTENTIOMETER_REVOLUTIONS * (constants.SCREW_TO_POT_RATIO * constants.SCREW_PITCH)) / (32768.0 * 1000.0));
statuses.healthStatus(
    isGood := position.statuses.healthStatus.isGood,
    hasWarning := position.statuses.healthStatus.hasWarning);

          

{attribute 'TcRpcEnable' := '1'}
METHOD _log : BOOL
  VAR_INPUT
    name : STRING;  (* Name of this function block instance *)
  END_VAR
  VAR_IN_OUT
    buffer : LogBuffer;  (* Buffer to write all logging to *)
  END_VAR
  VAR
    subBuffer : LogBuffer;  (* Temporary buffer to write logging by parts (sub-statemachines) to *)
  END_VAR
                  LOGGER(
    name := name,
    actualStatus := THIS^.actualStatus,
    previousStatus := THIS^.previousStatus,
    buffer := buffer,
    subBuffer := subBuffer,
    pHealthStatus := ADR(THIS^.statuses.healthStatus));

                
END_METHOD
END_FUNCTION_BLOCK

FUNCTION_BLOCK SM_M2TiltXAxis
  VAR_INPUT
    {attribute 'OPC.UA.DA' := '1'}
    {attribute 'OPC.UA.DA.Access' := '1'}
    position : LinearPositionMeasurement16;  (* Actual position of the axis *)
    {attribute 'OPC.UA.DA' := '1'}
    {attribute 'OPC.UA.DA.Access' := '1'}
    backlashLifted : BOOL;  (* TRUE if the backlash was previously lifted *)
    {attribute 'OPC.UA.DA' := '1'}
    {attribute 'OPC.UA.DA.Access' := '1'}
    powered : BOOL;  (* TRUE if the axis is powered *)
  END_VAR
  VAR_OUTPUT
    {attribute 'OPC.UA.DA' := '1'}
    {attribute 'OPC.UA.DA.Access' := '1'}
    actualStatus : STRING;  (* Current status description *)
    previousStatus : STRING;  (* Previous status description *)
    {attribute 'OPC.UA.DA' := '1'}
    {attribute 'OPC.UA.DA.Access' := '1'}
    constants : M2ConstantsTiltX;  (* Some constants particular for this axis *)
    statuses : M2TiltXAxisStatuses;  (* Statuses of the state machine *)
  END_VAR
  VAR_IN_OUT
    {attribute 'OPC.UA.DA' := '0'}
    config : M2Config;  (* The general M2 config *)
    {attribute 'OPC.UA.DA' := '0'}
    axisConfig : M2PotentiometerAxisConfig;  (* The config particular for this axis *)
  END_VAR

            position(
    config := axisConfig.general.measurement,
    conversionFactor := (constants.POTENTIOMETER_REVOLUTIONS * (constants.SCREW_TO_POT_RATIO * constants.SCREW_PITCH)) / (32768.0 * 1000.0));
statuses.healthStatus(
    isGood := position.statuses.healthStatus.isGood,
    hasWarning := position.statuses.healthStatus.hasWarning);

          

{attribute 'TcRpcEnable' := '1'}
METHOD _log : BOOL
  VAR_INPUT
    name : STRING;  (* Name of this function block instance *)
  END_VAR
  VAR_IN_OUT
    buffer : LogBuffer;  (* Buffer to write all logging to *)
  END_VAR
  VAR
    subBuffer : LogBuffer;  (* Temporary buffer to write logging by parts (sub-statemachines) to *)
  END_VAR
                  LOGGER(
    name := name,
    actualStatus := THIS^.actualStatus,
    previousStatus := THIS^.previousStatus,
    buffer := buffer,
    subBuffer := subBuffer,
    pHealthStatus := ADR(THIS^.statuses.healthStatus));

                
END_METHOD
END_FUNCTION_BLOCK

FUNCTION_BLOCK SM_M2TiltYAxis
  VAR_INPUT
    {attribute 'OPC.UA.DA' := '1'}
    {attribute 'OPC.UA.DA.Access' := '1'}
    position : LinearPositionMeasurement16;  (* Actual position of the axis *)
    {attribute 'OPC.UA.DA' := '1'}
    {attribute 'OPC.UA.DA.Access' := '1'}
    backlashLifted : BOOL;  (* TRUE if the backlash was previously lifted *)
    {attribute 'OPC.UA.DA' := '1'}
    {attribute 'OPC.UA.DA.Access' := '1'}
    powered : BOOL;  (* TRUE if the axis is powered *)
  END_VAR
  VAR_OUTPUT
    {attribute 'OPC.UA.DA' := '1'}
    {attribute 'OPC.UA.DA.Access' := '1'}
    actualStatus : STRING;  (* Current status description *)
    previousStatus : STRING;  (* Previous status description *)
    {attribute 'OPC.UA.DA' := '1'}
    {attribute 'OPC.UA.DA.Access' := '1'}
    constants : M2ConstantsTiltY;  (* Some constants particular for this axis *)
    statuses : M2TiltYAxisStatuses;  (* Statuses of the state machine *)
  END_VAR
  VAR_IN_OUT
    {attribute 'OPC.UA.DA' := '0'}
    config : M2Config;  (* The general M2 config *)
    {attribute 'OPC.UA.DA' := '0'}
    axisConfig : M2PotentiometerAxisConfig;  (* The config particular for this axis *)
  END_VAR

            position(
    config := axisConfig.general.measurement,
    conversionFactor := (constants.POTENTIOMETER_REVOLUTIONS * (constants.SCREW_TO_POT_RATIO * constants.SCREW_PITCH)) / (32768.0 * 1000.0));
statuses.healthStatus(
    isGood := position.statuses.healthStatus.isGood,
    hasWarning := position.statuses.healthStatus.hasWarning);

          

{attribute 'TcRpcEnable' := '1'}
METHOD _log : BOOL
  VAR_INPUT
    name : STRING;  (* Name of this function block instance *)
  END_VAR
  VAR_IN_OUT
    buffer : LogBuffer;  (* Buffer to write all logging to *)
  END_VAR
  VAR
    subBuffer : LogBuffer;  (* Temporary buffer to write logging by parts (sub-statemachines) to *)
  END_VAR
                  LOGGER(
    name := name,
    actualStatus := THIS^.actualStatus,
    previousStatus := THIS^.previousStatus,
    buffer := buffer,
    subBuffer := subBuffer,
    pHealthStatus := ADR(THIS^.statuses.healthStatus));

                
END_METHOD
END_FUNCTION_BLOCK

FUNCTION_BLOCK SM_M2ZAxis
  VAR_INPUT
    {attribute 'OPC.UA.DA' := '1'}
    {attribute 'OPC.UA.DA.Access' := '1'}
    position : LinearPositionMeasurementU32;  (* Actual position of the axis *)
    {attribute 'OPC.UA.DA' := '1'}
    {attribute 'OPC.UA.DA.Access' := '1'}
    backlashLifted : BOOL;  (* TRUE if the backlash was previously lifted *)
    {attribute 'OPC.UA.DA' := '1'}
    {attribute 'OPC.UA.DA.Access' := '1'}
    powered : BOOL;  (* TRUE if the axis is powered *)
    {attribute 'OPC.UA.DA' := '1'}
    {attribute 'OPC.UA.DA.Access' := '1'}
    isEnabled : BOOL;  (* TRUE if the Z axis control is enabled, FALSE if not *)
  END_VAR
  VAR_OUTPUT
    {attribute 'OPC.UA.DA' := '1'}
    {attribute 'OPC.UA.DA.Access' := '1'}
    actualStatus : STRING;  (* Current status description *)
    previousStatus : STRING;  (* Previous status description *)
    {attribute 'OPC.UA.DA' := '1'}
    {attribute 'OPC.UA.DA.Access' := '1'}
    constants : M2ConstantsZ;  (* Some constants particular for this axis *)
    statuses : M2ZAxisStatuses;  (* Statuses of the state machine *)
    parts : M2ZAxisParts;  (* Parts of the state machine *)
  END_VAR
  VAR_IN_OUT
    {attribute 'OPC.UA.DA' := '0'}
    config : M2Config;  (* The general M2 config *)
    {attribute 'OPC.UA.DA' := '0'}
    axisConfig : M2ZAxisConfig;  (* The config particular for this axis *)
  END_VAR

            position(
    rawValue := parts.encoder.counterValue,
    error := parts.encoder.dataError OR (parts.encoder.frameError OR (parts.encoder.powerFailure OR parts.encoder.syncError)),
    config := axisConfig.general.measurement,
    conversionFactor := (constants.SCREW_TO_ENC_RATIO * constants.SCREW_PITCH) / (8192.0 * 1000.0));
parts.highSpeed( isEnabled := isEnabled );
parts.encoder();
statuses.healthStatus(
    isGood := position.statuses.healthStatus.isGood AND parts.encoder.statuses.healthStatus.isGood,
    hasWarning := position.statuses.healthStatus.hasWarning OR parts.encoder.statuses.healthStatus.hasWarning);

          

{attribute 'TcRpcEnable' := '1'}
METHOD _log : BOOL
  VAR_INPUT
    name : STRING;  (* Name of this function block instance *)
  END_VAR
  VAR_IN_OUT
    buffer : LogBuffer;  (* Buffer to write all logging to *)
  END_VAR
  VAR
    subBuffer : LogBuffer;  (* Temporary buffer to write logging by parts (sub-statemachines) to *)
  END_VAR
                  THIS^.parts.highSpeed._log(
    name := 'highSpeed',
    buffer := subBuffer);
THIS^.parts.encoder._log(
    name := 'encoder',
    buffer := subBuffer);
LOGGER(
    name := name,
    actualStatus := THIS^.actualStatus,
    previousStatus := THIS^.previousStatus,
    buffer := buffer,
    subBuffer := subBuffer,
    pHealthStatus := ADR(THIS^.statuses.healthStatus));

                
END_METHOD
END_FUNCTION_BLOCK

FUNCTION_BLOCK SM_M2MoveStepsProcedure
  VAR_INPUT
    {attribute 'OPC.UA.DA' := '1'}
    {attribute 'OPC.UA.DA.Access' := '1'}
    state : M2MoveProcedureStates;  (* New state, to be set by the manual implementation *)
    {attribute 'OPC.UA.DA' := '1'}
    {attribute 'OPC.UA.DA.Access' := '1'}
    actualCounterValue AT %I* : UDINT;  (* Actual counter value *)
    {attribute 'OPC.UA.DA' := '1'}
    {attribute 'OPC.UA.DA.Access' := '1'}
    stepsRemaining : UDINT;  (* Number of steps remaining *)
  END_VAR
  VAR_OUTPUT
    {attribute 'OPC.UA.DA' := '1'}
    {attribute 'OPC.UA.DA.Access' := '1'}
    actualStatus : STRING;  (* Current status description *)
    previousStatus : STRING;  (* Previous status description *)
    statuses : M2MoveStepsProcedureStatuses;  (* Statuses of the state machine *)
  END_VAR
  VAR_IN_OUT
    {attribute 'OPC.UA.DA' := '0'}
    powerOn : Process;
    {attribute 'OPC.UA.DA' := '0'}
    x : M2XAxis;
    {attribute 'OPC.UA.DA' := '0'}
    y : M2YAxis;
    {attribute 'OPC.UA.DA' := '0'}
    z : M2ZAxis;
    {attribute 'OPC.UA.DA' := '0'}
    tiltX : M2TiltXAxis;
    {attribute 'OPC.UA.DA' := '0'}
    tiltY : M2TiltYAxis;
    {attribute 'OPC.UA.DA' := '0'}
    multiplexer : M2Multiplexer;
    {attribute 'OPC.UA.DA' := '0'}
    config : M2Config;
  END_VAR

            statuses.busyStatus( isBusy := NOT((state = M2MoveProcedureStates.IDLE) OR ((state = M2MoveProcedureStates.ABORTED) OR (state = M2MoveProcedureStates.ERROR))) );
statuses.healthStatus(
    isGood := NOT(state = M2MoveProcedureStates.ERROR),
    hasWarning := state = M2MoveProcedureStates.ABORTED);

          

{attribute 'TcRpcEnable' := '1'}
METHOD _log : BOOL
  VAR_INPUT
    name : STRING;  (* Name of this function block instance *)
  END_VAR
  VAR_IN_OUT
    buffer : LogBuffer;  (* Buffer to write all logging to *)
  END_VAR
  VAR
    subBuffer : LogBuffer;  (* Temporary buffer to write logging by parts (sub-statemachines) to *)
  END_VAR
                  LOGGER(
    name := name,
    actualStatus := THIS^.actualStatus,
    previousStatus := THIS^.previousStatus,
    buffer := buffer,
    subBuffer := subBuffer,
    pHealthStatus := ADR(THIS^.statuses.healthStatus),
    pBusyStatus := ADR(THIS^.statuses.busyStatus));

                
END_METHOD
END_FUNCTION_BLOCK

FUNCTION_BLOCK SM_M2MovePositionProcedure
  VAR_INPUT
    {attribute 'OPC.UA.DA' := '1'}
    {attribute 'OPC.UA.DA.Access' := '1'}
    state : M2MoveProcedureStates;  (* New state, to be set by the manual implementation *)
  END_VAR
  VAR_OUTPUT
    {attribute 'OPC.UA.DA' := '1'}
    {attribute 'OPC.UA.DA.Access' := '1'}
    actualStatus : STRING;  (* Current status description *)
    previousStatus : STRING;  (* Previous status description *)
    statuses : M2MovePositionProcedureStatuses;  (* Statuses of the state machine *)
  END_VAR
  VAR_IN_OUT
    {attribute 'OPC.UA.DA' := '0'}
    powerOn : Process;
    {attribute 'OPC.UA.DA' := '0'}
    x : M2XAxis;
    {attribute 'OPC.UA.DA' := '0'}
    y : M2YAxis;
    {attribute 'OPC.UA.DA' := '0'}
    z : M2ZAxis;
    {attribute 'OPC.UA.DA' := '0'}
    tiltX : M2TiltXAxis;
    {attribute 'OPC.UA.DA' := '0'}
    tiltY : M2TiltYAxis;
    {attribute 'OPC.UA.DA' := '0'}
    multiplexer : M2Multiplexer;
    {attribute 'OPC.UA.DA' := '0'}
    moveStepsProcedure : M2MoveStepsProcedure;
    {attribute 'OPC.UA.DA' := '0'}
    config : M2Config;
  END_VAR

            statuses.busyStatus( isBusy := NOT((state = M2MoveProcedureStates.IDLE) OR ((state = M2MoveProcedureStates.ABORTED) OR (state = M2MoveProcedureStates.ERROR))) );
statuses.healthStatus(
    isGood := NOT(state = M2MoveProcedureStates.ERROR),
    hasWarning := state = M2MoveProcedureStates.ABORTED);

          

{attribute 'TcRpcEnable' := '1'}
METHOD _log : BOOL
  VAR_INPUT
    name : STRING;  (* Name of this function block instance *)
  END_VAR
  VAR_IN_OUT
    buffer : LogBuffer;  (* Buffer to write all logging to *)
  END_VAR
  VAR
    subBuffer : LogBuffer;  (* Temporary buffer to write logging by parts (sub-statemachines) to *)
  END_VAR
                  LOGGER(
    name := name,
    actualStatus := THIS^.actualStatus,
    previousStatus := THIS^.previousStatus,
    buffer := buffer,
    subBuffer := subBuffer,
    pHealthStatus := ADR(THIS^.statuses.healthStatus),
    pBusyStatus := ADR(THIS^.statuses.busyStatus));

                
END_METHOD
END_FUNCTION_BLOCK

FUNCTION_BLOCK M2SelectAxisProcess EXTENDS BaseProcess
  VAR_INPUT
    {attribute 'OPC.UA.DA' := '1'}
    set : M2SelectAxisProcessArgs;  (* Arguments to be set, before writing do_request TRUE *)
  END_VAR
  VAR_OUTPUT
    {attribute 'OPC.UA.DA' := '1'}
    {attribute 'OPC.UA.DA.Access' := '1'}
    get : M2SelectAxisProcessArgs;  (* Arguments in use by the process, if do_request was accepted *)
  END_VAR

            IF do_request THEN
    do_request_result := request( axis := set.axis );
    do_request := FALSE;
END_IF;
SUPER^();

          

{attribute 'TcRpcEnable' := '1'}
METHOD start
  VAR_INPUT
    axis : M2Axes;  (* The axis to select *)
  END_VAR
                  THIS^.get.axis := axis;
THIS^.statuses.busyStatus( isBusy := TRUE );
THIS^.statuses.healthStatus( isGood := TRUE );

                
END_METHOD

{attribute 'TcRpcEnable' := '1'}
METHOD request : RequestResults
  VAR_INPUT
    axis : M2Axes;  (* The axis to select *)
  END_VAR
                  IF THIS^.statuses.enabledStatus.enabled THEN
    THIS^.start( axis := axis );
    request := RequestResults.ACCEPTED;
ELSE
    request := RequestResults.REJECTED;
END_IF;

                
END_METHOD
END_FUNCTION_BLOCK

FUNCTION_BLOCK M2MoveProcess EXTENDS BaseProcess
  VAR_INPUT
    {attribute 'OPC.UA.DA' := '1'}
    set : M2MoveProcessArgs;  (* Arguments to be set, before writing do_request TRUE *)
  END_VAR
  VAR_OUTPUT
    {attribute 'OPC.UA.DA' := '1'}
    {attribute 'OPC.UA.DA.Access' := '1'}
    get : M2MoveProcessArgs;  (* Arguments in use by the process, if do_request was accepted *)
  END_VAR

            IF do_request THEN
    do_request_result := request(
    axis := set.axis,
    position := set.position);
    do_request := FALSE;
END_IF;
SUPER^();

          

{attribute 'TcRpcEnable' := '1'}
METHOD start
  VAR_INPUT
    axis : M2Axes;  (* The axis to move *)
    position : LREAL;  (* Move to a certain position in millimeters *)
  END_VAR
                  THIS^.get.axis := axis;
THIS^.get.position := position;
THIS^.statuses.busyStatus( isBusy := TRUE );
THIS^.statuses.healthStatus( isGood := TRUE );

                
END_METHOD

{attribute 'TcRpcEnable' := '1'}
METHOD request : RequestResults
  VAR_INPUT
    axis : M2Axes;  (* The axis to move *)
    position : LREAL;  (* Move to a certain position in millimeters *)
  END_VAR
                  IF THIS^.statuses.enabledStatus.enabled THEN
    THIS^.start(
        axis := axis,
        position := position);
    request := RequestResults.ACCEPTED;
ELSE
    request := RequestResults.REJECTED;
END_IF;

                
END_METHOD
END_FUNCTION_BLOCK

FUNCTION_BLOCK M2MoveStepsProcess EXTENDS BaseProcess
  VAR_INPUT
    {attribute 'OPC.UA.DA' := '1'}
    set : M2MoveStepsProcessArgs;  (* Arguments to be set, before writing do_request TRUE *)
  END_VAR
  VAR_OUTPUT
    {attribute 'OPC.UA.DA' := '1'}
    {attribute 'OPC.UA.DA.Access' := '1'}
    get : M2MoveStepsProcessArgs;  (* Arguments in use by the process, if do_request was accepted *)
  END_VAR

            IF do_request THEN
    do_request_result := request(
    axis := set.axis,
    steps := set.steps,
    cw := set.cw,
    fast := set.fast);
    do_request := FALSE;
END_IF;
SUPER^();

          

{attribute 'TcRpcEnable' := '1'}
METHOD start
  VAR_INPUT
    axis : M2Axes;  (* The axis to move *)
    steps : UDINT;  (* Move a certain number of steps *)
    cw : BOOL;  (* True if the axis should be moved in CW (negative) direction *)
    fast : BOOL;  (* True if the axis should be moved fast (only used in case of Z-axis!) *)
  END_VAR
                  THIS^.get.axis := axis;
THIS^.get.steps := steps;
THIS^.get.cw := cw;
THIS^.get.fast := fast;
THIS^.statuses.busyStatus( isBusy := TRUE );
THIS^.statuses.healthStatus( isGood := TRUE );

                
END_METHOD

{attribute 'TcRpcEnable' := '1'}
METHOD request : RequestResults
  VAR_INPUT
    axis : M2Axes;  (* The axis to move *)
    steps : UDINT;  (* Move a certain number of steps *)
    cw : BOOL;  (* True if the axis should be moved in CW (negative) direction *)
    fast : BOOL;  (* True if the axis should be moved fast (only used in case of Z-axis!) *)
  END_VAR
                  IF THIS^.statuses.enabledStatus.enabled THEN
    THIS^.start(
        axis := axis,
        steps := steps,
        cw := cw,
        fast := fast);
    request := RequestResults.ACCEPTED;
ELSE
    request := RequestResults.REJECTED;
END_IF;

                
END_METHOD
END_FUNCTION_BLOCK

FUNCTION_BLOCK M2DoThermalFocusForStationPosition EXTENDS BaseProcess
  VAR_INPUT
    {attribute 'OPC.UA.DA' := '1'}
    set : M2DoThermalFocusForStationPositionArgs;  (* Arguments to be set, before writing do_request TRUE *)
  END_VAR
  VAR_OUTPUT
    {attribute 'OPC.UA.DA' := '1'}
    {attribute 'OPC.UA.DA.Access' := '1'}
    get : M2DoThermalFocusForStationPositionArgs;  (* Arguments in use by the process, if do_request was accepted *)
  END_VAR

            IF do_request THEN
    do_request_result := request( station := set.station );
    do_request := FALSE;
END_IF;
SUPER^();

          

{attribute 'TcRpcEnable' := '1'}
METHOD start
  VAR_INPUT
    station : M3PositionIDs;  (* The station numerical ID for which the thermal focus should be executed *)
  END_VAR
                  THIS^.get.station := station;
THIS^.statuses.busyStatus( isBusy := TRUE );
THIS^.statuses.healthStatus( isGood := TRUE );

                
END_METHOD

{attribute 'TcRpcEnable' := '1'}
METHOD request : RequestResults
  VAR_INPUT
    station : M3PositionIDs;  (* The station numerical ID for which the thermal focus should be executed *)
  END_VAR
                  IF THIS^.statuses.enabledStatus.enabled THEN
    THIS^.start( station := station );
    request := RequestResults.ACCEPTED;
ELSE
    request := RequestResults.REJECTED;
END_IF;

                
END_METHOD
END_FUNCTION_BLOCK

FUNCTION_BLOCK M2DoThermalFocusForStationName EXTENDS BaseProcess
  VAR_INPUT
    {attribute 'OPC.UA.DA' := '1'}
    set : M2DoThermalFocusForStationNameArgs;  (* Arguments to be set, before writing do_request TRUE *)
  END_VAR
  VAR_OUTPUT
    {attribute 'OPC.UA.DA' := '1'}
    {attribute 'OPC.UA.DA.Access' := '1'}
    get : M2DoThermalFocusForStationNameArgs;  (* Arguments in use by the process, if do_request was accepted *)
  END_VAR

            IF do_request THEN
    do_request_result := request( station := set.station );
    do_request := FALSE;
END_IF;
SUPER^();

          

{attribute 'TcRpcEnable' := '1'}
METHOD start
  VAR_INPUT
    station : STRING;  (* The configured station name, for which the thermal focus should be executed *)
  END_VAR
                  THIS^.get.station := station;
THIS^.statuses.busyStatus( isBusy := TRUE );
THIS^.statuses.healthStatus( isGood := TRUE );

                
END_METHOD

{attribute 'TcRpcEnable' := '1'}
METHOD request : RequestResults
  VAR_INPUT
    station : STRING;  (* The configured station name, for which the thermal focus should be executed *)
  END_VAR
                  IF THIS^.statuses.enabledStatus.enabled THEN
    THIS^.start( station := station );
    request := RequestResults.ACCEPTED;
ELSE
    request := RequestResults.REJECTED;
END_IF;

                
END_METHOD
END_FUNCTION_BLOCK
